# EPICS autosave request: softGlueApp/Db/softGlue_FPGAContent_Encoder_settings.req
# up/dn counters
file UpDnCntr_settings.req P=$(P),H=$(H),N=1
file UpDnCntr_settings.req P=$(P),H=$(H),N=2
file QuadDec_settings.req P=$(P),H=$(H),N=1
file QuadDec_settings.req P=$(P),H=$(H),N=2
